// Mitsubishi GX Works2 project: 20151029(パラメータ設定)   PLC: Q03UDV

PROGRAM P1
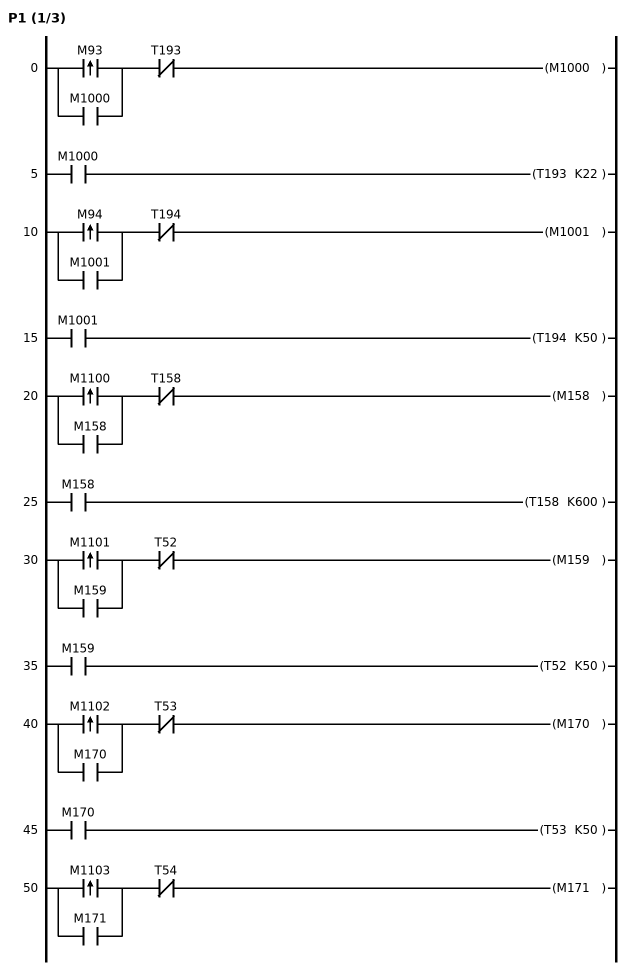
0     LDP     M93
      OR      M1000
      ANI     T193
      OUT     M1000
5     LD      M1000
      OUT     T193 K22
10    LDP     M94
      OR      M1001
      ANI     T194
      OUT     M1001
15    LD      M1001
      OUT     T194 K50
20    LDP     M1100
      OR      M158
      ANI     T158
      OUT     M158
25    LD      M158
      OUT     T158 K600
30    LDP     M1101
      OR      M159
      ANI     T52
      OUT     M159
35    LD      M159
      OUT     T52 K50
40    LDP     M1102
      OR      M170
      ANI     T53
      OUT     M170
45    LD      M170
      OUT     T53 K50
50    LDP     M1103
      OR      M171
      ANI     T54
      OUT     M171
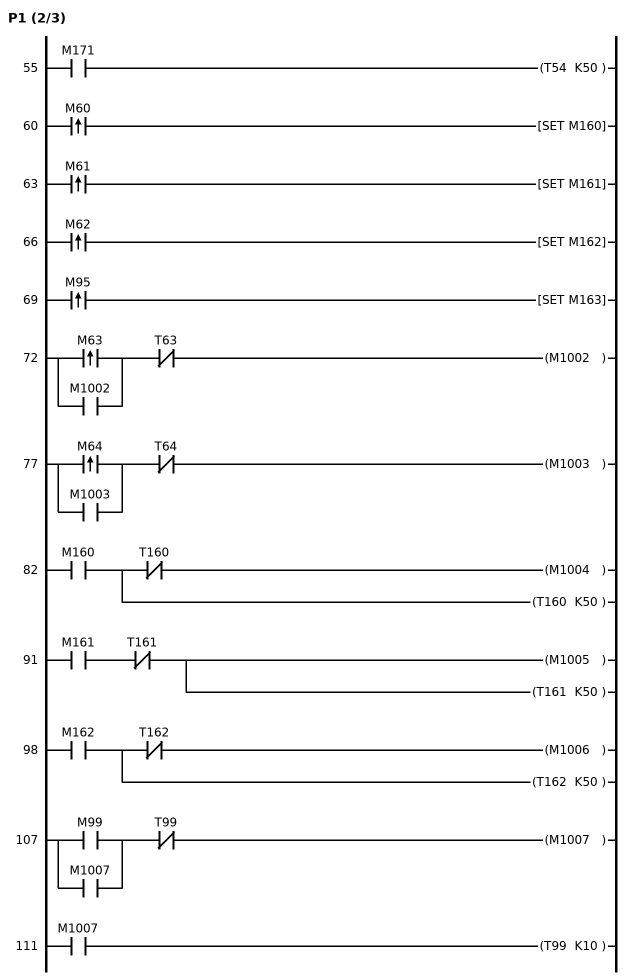
55    LD      M171
      OUT     T54 K50
60    LDP     M60
      SET     M160
63    LDP     M61
      SET     M161
66    LDP     M62
      SET     M162
69    LDP     M95
      SET     M163
72    LDP     M63
      OR      M1002
      ANI     T63
      OUT     M1002
77    LDP     M64
      OR      M1003
      ANI     T64
      OUT     M1003
82    LD      M160
      MPS
      ANI     T160
      OUT     M1004
      MPP
      OUT     T160 K50
91    LD      M161
      ANI     T161
      OUT     M1005
      OUT     T161 K50
98    LD      M162
      MPS
      ANI     T162
      OUT     M1006
      MPP
      OUT     T162 K50
107   LD      M99
      OR      M1007
      ANI     T99
      OUT     M1007
111   LD      M1007
      OUT     T99 K10
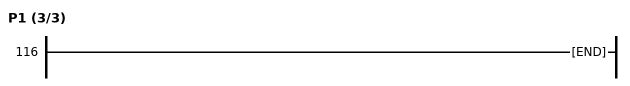
116   END
END_PROGRAM
